FUNCTION_BLOCK FB_TareaGeneral

VAR_INPUT
    // SFC-Flags
    SFCPause: BOOL;
    SFCReset: BOOL;
    
    // Parametros de control de la estacion
    CicloACiclo: BOOL;    

    // Parametros de control de la tarea
    UnidadesSolicitadas: UINT := 1; 
    TipoUnidadSolicitada: BYTE; // 0 = rodamiento bajo; 1 = rodamiento alto

    // Parametros de tiempo
    TpoCintaRetenedor: TIME := T#1S;
    TpoPaleEntrada: TIME := T#400MS;
    TpoPaleSalida: TIME := T#1s;
    TpoPaleTransferencia: TIME := T#1S;
    
    TpoPrensaHidraulico: TIME := T#2s;
    TpoPrensaProtector: TIME := T#2S; 
	
    
	MedidorAltura AT %I* : UINT;
    PulsadorEmergencia AT %I* : BOOL;
    SelectorManual AT %I* : BOOL;
    PulsadorMarcha AT %I* : BOOL;
    PulsadorParada AT %I* : BOOL;
    EstacionConectada AT %I* : BOOL;
    PresenciaPale AT %I* : BOOL;
    CodigoPaleBit0 AT %I* : BOOL;
    CodigoPaleBit1 AT  %I* : BOOL;
    
    CodigoPaleBit2 AT %I* : BOOL;
    CargadorDetras AT %I* : BOOL;
    CargadorDelante AT %I* : BOOL;
    CargadorArriba AT %I* : BOOL;
    CargadorAbajo AT %I* : BOOL;
    PlatoEmpujadorDetras AT %I* : BOOL;
    RechazadorDetras AT %I* : BOOL;
    RechazadorDelante AT %I* : BOOL;
    RechazadorArriba AT %I* : BOOL;
    
    RechazadorVacio AT %I* : BOOL;
    DescargadorDetras AT %I* : BOOL;
    DescargadorDelante AT %I* : BOOL;
    DescargadorArriba AT %I* : BOOL;
    DescargadorAbajo AT %I* : BOOL;
    AlimentadorDelante AT %I* : BOOL;
    DetectorInductivo AT %I* : BOOL;
    DetectorFotoelectrico AT %I* : BOOL;
    VolteadorArriba AT %I* : BOOL;
    VolteadorAbajo AT %I* : BOOL;
    VolteadorDetras AT %I* : BOOL;
    VoteadorDelante AT %I* : BOOL;   
END_VAR
VAR_OUTPUT
    // Parametros de; estado de la estacion
    CondicionInicial: BOOL:=TRUE;
    CondicionMarcha: BOOL:=TRUE;
    CodigoPale: BYTE;  
	Medir: BOOL := FALSE;
    
    // Parametros de control de la tarea 
    UnidadesPendientes: UINT;
    UnidadesRealizadas: UINT;
    

	
	DesconectaEstacion AT %Q* : BOOL;
    LamparaAlarma AT %Q* : BOOL;
    LamparaMarcha AT %Q* : BOOL;
    LamparaMaterial AT %Q* : BOOL;
    CintaActiva AT %Q* : BOOL;
    CintaInvierte AT %Q* : BOOL;
    RetenedorBaja AT %Q* : BOOL;
    
    AvisadorSonoro AT %Q* : BOOL;
  	CargadorAvanza AT %Q* : BOOL;
    CargadorBaja AT %Q* : BOOL;
    CargadorCierra AT %Q* : BOOL;
    PlatoEmpujadorAvanza AT %Q* : BOOL;
    PlatoRetenedorAtras AT %Q* : BOOL;
    RechazadorAvanza AT %Q* : BOOL;
    RechazadorRetrocede AT %Q* : BOOL;
    RechazadorBaja AT %Q* : BOOL;
    
    RechazadorSucciona AT %Q* : BOOL;
    DescargadorAvanza AT %Q* : BOOL;
    DescargadorBaja AT %Q* : BOOL;
    DescargadorCierra AT %Q* : BOOL;
    AlimentadorAvanza AT %Q* : BOOL;
    MedidorBaja AT %Q* : BOOL;
    VolteadorBaja AT %Q* : BOOL;
    VolteadorGira AT %Q* : BOOL;
    VolteadorCierra AT %Q* : BOOL;
END_VAR
VAR
    // Tapas: (METALICAS, BLANCAS, NEGRAS, ALTAS, BAJAS);
    Tapas : ARRAY[0..7] OF ST_POSICION;
    TapaAuxRot : ST_POSICION; 
    CLK: FB_Clock;
    
    TapaDeseada : ST_TAPA;
    NumPiezasDes: UINT;
    cont: UINT;
  
END_VAR

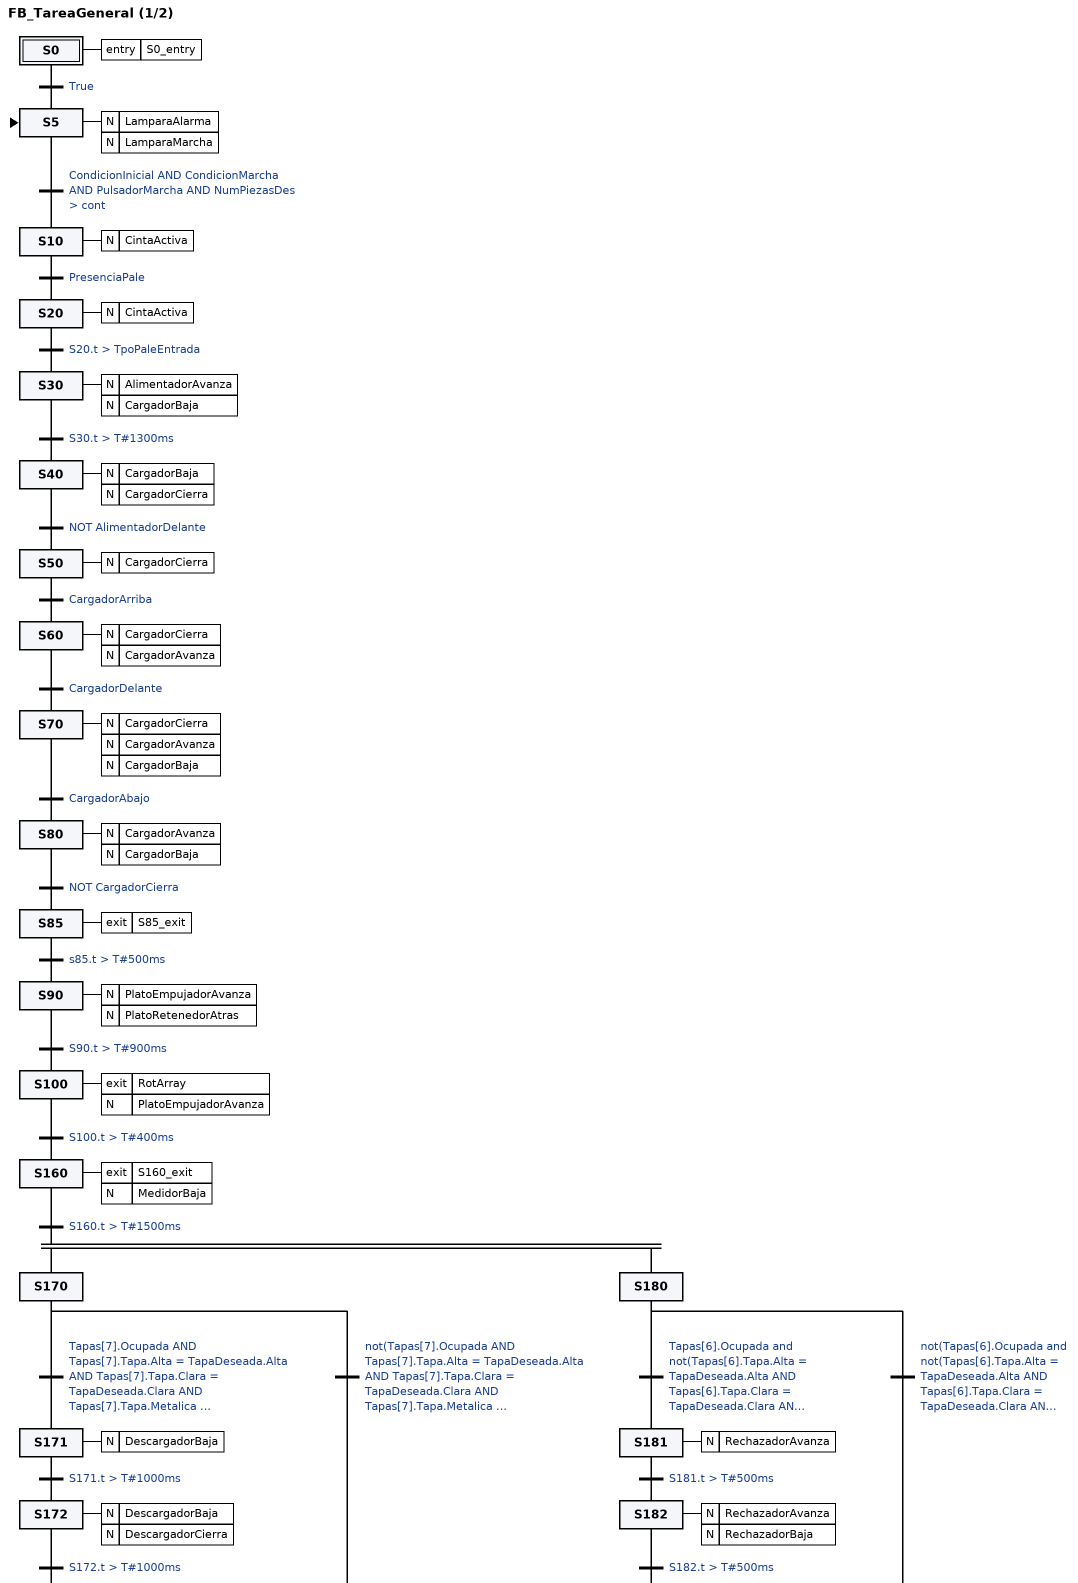
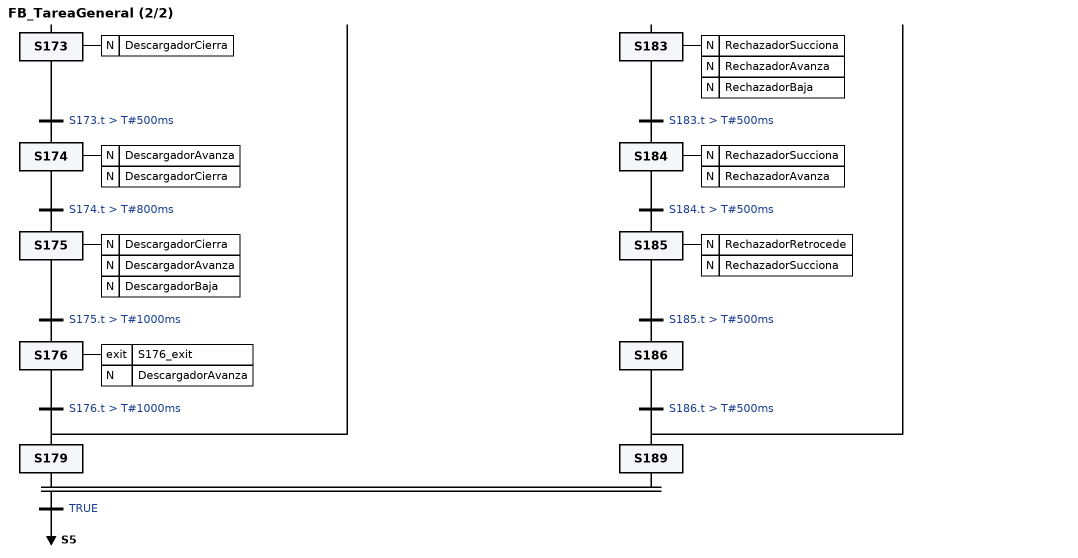
INITIAL_STEP S0:
    S0_entry(P1);  // entry action
END_STEP
TRANSITION FROM S0 TO S5
    := True;
END_TRANSITION
STEP S5:
    LamparaAlarma(N);
    LamparaMarcha(N);
END_STEP
TRANSITION FROM S5 TO S10
    := CondicionInicial AND CondicionMarcha AND PulsadorMarcha AND NumPiezasDes > cont;
END_TRANSITION
STEP S10:
    CintaActiva(N);
END_STEP
TRANSITION FROM S10 TO S20
    := PresenciaPale;
END_TRANSITION
STEP S20:
    CintaActiva(N);
END_STEP
TRANSITION FROM S20 TO S30
    := S20.t > TpoPaleEntrada;
END_TRANSITION
STEP S30:
    AlimentadorAvanza(N);
    CargadorBaja(N);
END_STEP
TRANSITION FROM S30 TO S40
    := S30.t > T#1300ms;
END_TRANSITION
STEP S40:
    CargadorBaja(N);
    CargadorCierra(N);
END_STEP
TRANSITION FROM S40 TO S50
    := NOT AlimentadorDelante;
END_TRANSITION
STEP S50:
    CargadorCierra(N);
END_STEP
TRANSITION FROM S50 TO S60
    := CargadorArriba;
END_TRANSITION
STEP S60:
    CargadorCierra(N);
    CargadorAvanza(N);
END_STEP
TRANSITION FROM S60 TO S70
    := CargadorDelante;
END_TRANSITION
STEP S70:
    CargadorCierra(N);
    CargadorAvanza(N);
    CargadorBaja(N);
END_STEP
TRANSITION FROM S70 TO S80
    := CargadorAbajo;
END_TRANSITION
STEP S80:
    CargadorAvanza(N);
    CargadorBaja(N);
END_STEP
TRANSITION FROM S80 TO S85
    := NOT CargadorCierra;
END_TRANSITION
STEP S85:
    S85_exit(P0);  // exit action
END_STEP
TRANSITION FROM S85 TO S90
    := s85.t > T#500ms;
END_TRANSITION
STEP S90:
    PlatoEmpujadorAvanza(N);
    PlatoRetenedorAtras(N);
END_STEP
TRANSITION FROM S90 TO S100
    := S90.t > T#900ms;
END_TRANSITION
STEP S100:
    RotArray(P0);  // exit action
    PlatoEmpujadorAvanza(N);
END_STEP
TRANSITION FROM S100 TO S160
    := S100.t > T#400ms;
END_TRANSITION
STEP S160:
    S160_exit(P0);  // exit action
    MedidorBaja(N);
END_STEP
TRANSITION FROM S160 TO (S170, S180)
    := S160.t > T#1500ms;
END_TRANSITION
STEP S170:
END_STEP
TRANSITION FROM S170 TO S171
    := Tapas[7].Ocupada AND Tapas[7].Tapa.Alta = TapaDeseada.Alta AND Tapas[7].Tapa.Clara = TapaDeseada.Clara AND Tapas[7].Tapa.Metalica = TapaDeseada.Metalica;
END_TRANSITION
STEP S171:
    DescargadorBaja(N);
END_STEP
TRANSITION FROM S171 TO S172
    := S171.t > T#1000ms;
END_TRANSITION
STEP S172:
    DescargadorBaja(N);
    DescargadorCierra(N);
END_STEP
TRANSITION FROM S172 TO S173
    := S172.t > T#1000ms;
END_TRANSITION
STEP S173:
    DescargadorCierra(N);
END_STEP
TRANSITION FROM S173 TO S174
    := S173.t > T#500ms;
END_TRANSITION
STEP S174:
    DescargadorAvanza(N);
    DescargadorCierra(N);
END_STEP
TRANSITION FROM S174 TO S175
    := S174.t > T#800ms;
END_TRANSITION
STEP S175:
    DescargadorCierra(N);
    DescargadorAvanza(N);
    DescargadorBaja(N);
END_STEP
TRANSITION FROM S175 TO S176
    := S175.t > T#1000ms;
END_TRANSITION
STEP S176:
    S176_exit(P0);  // exit action
    DescargadorAvanza(N);
END_STEP
TRANSITION FROM S176 TO S179
    := S176.t > T#1000ms;
END_TRANSITION
TRANSITION FROM S170 TO S179
    := not(Tapas[7].Ocupada AND Tapas[7].Tapa.Alta = TapaDeseada.Alta AND Tapas[7].Tapa.Clara = TapaDeseada.Clara AND Tapas[7].Tapa.Metalica = TapaDeseada.Metalica);
END_TRANSITION
STEP S179:
END_STEP
STEP S180:
END_STEP
TRANSITION FROM S180 TO S181
    := Tapas[6].Ocupada and not(Tapas[6].Tapa.Alta = TapaDeseada.Alta AND Tapas[6].Tapa.Clara = TapaDeseada.Clara AND Tapas[6].Tapa.Metalica = TapaDeseada.Metalica);
END_TRANSITION
STEP S181:
    RechazadorAvanza(N);
END_STEP
TRANSITION FROM S181 TO S182
    := S181.t > T#500ms;
END_TRANSITION
STEP S182:
    RechazadorAvanza(N);
    RechazadorBaja(N);
END_STEP
TRANSITION FROM S182 TO S183
    := S182.t > T#500ms;
END_TRANSITION
STEP S183:
    RechazadorSucciona(N);
    RechazadorAvanza(N);
    RechazadorBaja(N);
END_STEP
TRANSITION FROM S183 TO S184
    := S183.t > T#500ms;
END_TRANSITION
STEP S184:
    RechazadorSucciona(N);
    RechazadorAvanza(N);
END_STEP
TRANSITION FROM S184 TO S185
    := S184.t > T#500ms;
END_TRANSITION
STEP S185:
    RechazadorRetrocede(N);
    RechazadorSucciona(N);
END_STEP
TRANSITION FROM S185 TO S186
    := S185.t > T#500ms;
END_TRANSITION
STEP S186:
END_STEP
TRANSITION FROM S186 TO S189
    := S186.t > T#500ms;
END_TRANSITION
TRANSITION FROM S180 TO S189
    := not(Tapas[6].Ocupada and not(Tapas[6].Tapa.Alta = TapaDeseada.Alta AND Tapas[6].Tapa.Clara = TapaDeseada.Clara AND Tapas[6].Tapa.Metalica = TapaDeseada.Metalica));
END_TRANSITION
STEP S189:
END_STEP
TRANSITION FROM (S179, S189) TO S5
    := TRUE;
END_TRANSITION

ACTION RotArray:
TapaAuxRot := Tapas[7];
Tapas[7] := Tapas[6];
Tapas[6] := Tapas[5];
Tapas[5] := Tapas[4];
Tapas[4] := Tapas[3];
Tapas[3] := Tapas[2];
Tapas[2] := Tapas[1];
Tapas[1] := Tapas[0];
Tapas[0] := TapaAuxRot;
END_ACTION

ACTION S0_entry:
cont := 0;
Tapas[0].Ocupada := 0;
Tapas[1].Ocupada := 0;
Tapas[2].Ocupada := 0;
Tapas[3].Ocupada := 0;
Tapas[4].Ocupada := 0;
Tapas[5].Ocupada := 0;
Tapas[6].Ocupada := 0;
Tapas[7].Ocupada := 0;
END_ACTION

ACTION S160_exit:
Tapas[2].Tapa.Alta := (MedidorAltura <= 1300);
Tapas[3].Tapa.Clara := DetectorFotoelectrico;
Tapas[4].Tapa.Metalica := DetectorInductivo;
END_ACTION

ACTION S171_entry:

END_ACTION

ACTION S176_exit:
cont := cont + 1;
END_ACTION

ACTION S85_exit:
Tapas[0].Ocupada := TRUE;
END_ACTION

END_FUNCTION_BLOCK

(* stored: Version 1.1.0.1, ProductVersion 3.1.4024.12
   POU FB_TareaGeneral: Id {df13f857-ec23-424a-8bc1-2cda1ca9ee95}, SpecialFunc None
   Action RotArray: Id {d2258d71-d1ae-43c7-b4d8-bc3edbd917ec}
   Action S0_entry: Id {faf887e1-7e8f-4007-868f-2b755c57d673}
   Action S160_exit: Id {364aa1c2-2031-4277-9c42-436897932e92}
   Action S171_entry: Id {518da548-90d4-42bd-8d42-0e0def533d09}
   Action S176_exit: Id {a8a65394-50d3-4c9d-8346-fde83d0b8e2e}
   Action S85_exit: Id {c47f20e4-f986-407c-a5ec-7ebd72460b11} *)
